{attribute 'qualified_only'}
TYPE E_ClampCommand : (NONE := 0, CLAMP := 1, UNCLAMP := 2) DINT;
END_TYPE

(* stored: Version 1.1.0.1, ProductVersion 3.1.4024.12
   DUT E_ClampCommand: Id {04c4ad14-3a16-4fb7-a1ec-ee24b4f5b1e9} *)
